// TIA Portal V20 export
TYPE "typeEstopStatus"
// stored: Access Published, IsFailsafeCompliant true, Namespace Safety
   STRUCT
      mainOpEmoPressed : Bool;   // Main OP EMO Pressed
      unwinderCenterEmoPressed : Bool;   // Unwinder Center EMO Pressed
      jrOutPutEmoPressed : Bool;   // JR Output EMO Pressed
      anodeRearEmoPressed : Bool;   // Anode Rear EMO Pressed
      cathodeRearEmoPressed : Bool;   // Cathode Rear EMO Pressed
      pHmiEmoPressed : Bool;   // PHMI1 EMO Pressed
      ba10EmoPressed : Bool;   // CathodeReelcut EMO pressed
      ba15EmoPressed : Bool;   // AnodeReelcut EMO pressed
      ba30EmoPressed : Bool;   // Stacker1 EMO pressed
      ba60EmoPressed : Bool;   // Inspection EMO pressed
   END_STRUCT;
END_TYPE
